{region '#Template'}
	{attribute 'Category' := 'Universal'}
	{attribute 'Version' := '0.0.1.0'}
	{attribute 'Tags' := 'Universal, Sensor, BI'}
	{attribute 'Description' := 'BI	mit IO // BI with IO'}
{endregion}
FUNCTION_BLOCK FB_BA_SensorBinary_IO EXTENDS FB_BA_View
VAR_INPUT
END_VAR
VAR_INPUT CONSTANT
	Input					: FB_BA_BI_IO;		
END_VAR
VAR_OUTPUT
	bPresentValue			: BOOL;	
END_VAR
VAR
END_VAR

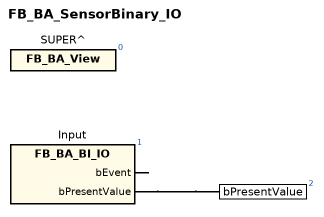
SUPER^(); // FB_BA_View
Input(); // FB_BA_BI_IO
bPresentValue := Input.bPresentValue;

METHOD FB_init : BOOL
VAR_INPUT
	bInitRetains : BOOL; // if TRUE, the retain variables are initialized (warm start / cold start)
	bInCopyCode : BOOL;  // if TRUE, the instance afterwards gets moved into the copy code (online change)
END_VAR
Input.iParent						:= THIS^;
Input.iLabel						:= LblUniFieldDevice.SensorBinary_Input;	
Input.sObjectName					:= '{Idx=01}';	
Input.sDeviceType					:= '';
Input.bEnOutOfService				:= FALSE;
Input.ePolarity						:= E_BA_Polarity.eReverse;
Input.sActiveText 					:= Texts.txtTriggered;
Input.sInactiveText 				:= Texts.txtNormal;
Input.nStateChangeCount				:= 0;
Input.nActiveTimeElapsed			:= 0;
Input.nEventClassID					:= EventClasses.AlarmTechnicalExtended;
Input.stTimeDelay.nToNormal			:= BA2_Param.nDefTimeDelay_ToNormal;
Input.stTimeDelay.nToAbnormal		:= BA2_Param.nDefTimeDelay_ToAbnormal;
Input.bAlarmValue					:= TRUE;
Input.bAcknowledgeRm				:= FALSE;		
Input.aEventTransitionText[1]		:= Texts.txtTriggered;
Input.aEventTransitionText[2]		:= Texts.txtError;
Input.aEventTransitionText[3]		:= Texts.txtNormal;
Input.bEventDetectionEnable			:= TRUE;
Input.eEnPlantLock					:= E_BA_LockPriority.eNoLock;
END_METHOD

END_FUNCTION_BLOCK

(* stored: Version 1.1.0.1, ProductVersion 3.1.4024.6
   POU FB_BA_SensorBinary_IO: Id {54eab52d-e324-4e4f-8b8d-c0e22b19b762}, SpecialFunc None
   Method FB_init: Id {2dbb9e34-6250-448e-8ddc-49479a7d4711} *)
